PROGRAM Alarmy
VAR
	Migacz: FB_Blink_S;
END_VAR


Migacz(Tv:=T#500MS , Q=> );

END_PROGRAM

(* stored: Version 1.1.0.1, ProductVersion 3.1.4024.15
   POU Alarmy: Id {8cd91d19-e7e8-47aa-8be1-a23412e084d2}, SpecialFunc None *)
